RoboDK station: Rib.rdk

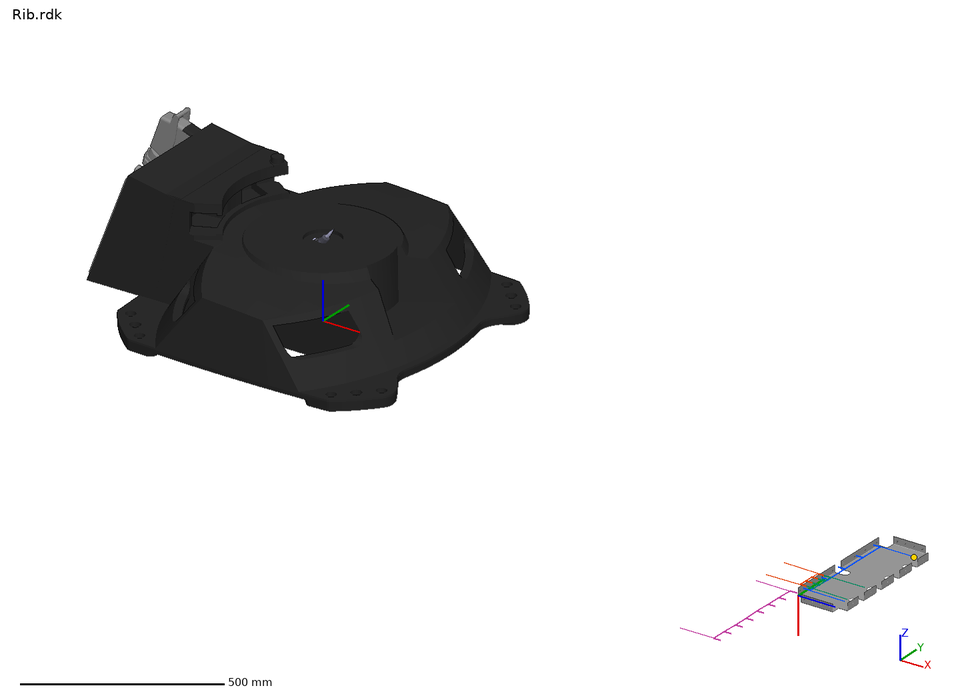
[picture v0: the station drawn from its stored meshes, robots at their saved joint values, targets as dots, program paths as lines]
Station Rib (saved by RoboDK 5.2.3). Poses are relative to the parent item; angles as X-Y-Z fixed-axis rotations.
  - frame KUKA KR 210 R2700 extra Base at (0, 0, 0) mm
    - robot KUKA KR 210 R2700 extra: 6 axes, payload 210 kg, reach 2696 mm, repeatability 0.06 mm, weight 1068 kg
        joint limits [-185, -140, -120, -350, -125, -350] to [185, -5, 155, 350, 125, 350]; home [0, -90, 90, 0, 0, 0]; saved at [-33.949, -82.089, 134.053, 57.76, 80.009, -97.195]
      - tool Spindle, TCP at (32, 0, 260) mm, rotated rx 0 ry 39 rz 0 deg, size 157.3 x 72 x 259.9 mm, geometry from Extracted Curve Point
  - frame Frame 2 at (1418.68, 0, -350) mm, rotated rx 0 ry 90 rz 0 deg
    - object rib-side at (0, 369, 0) mm, rotated rx 90 ry 0 rz 0 deg, 4 curves, geometry from Point 4
    - object rib-side at (0, -27, 0) mm, rotated rx 90 ry 0 rz 0 deg, 4 curves, geometry from Point 4
    - object rib-top at (0, 0, 146.5) mm, 5 curves, geometry from Point 5
    - object Rib at (0, 0, 0) mm, size 21.8 x 396 x 148.8 mm, geometry from Rib.stl
    - object rib-bot at (-21, 0, 0) mm, rotated rx 0 ry 0 rz 180 deg, 8 curves, geometry from Point 8
  - program target4 (36 instructions, listed below)
  - machining project Point settings: rotZ(0) | rotX(0)*rotY(0) | rotz(0) | onStart | onPathStart | onApproach | onPoint | onRetract | onFinish | SetRPM(%1) | SetTool(%1) | Extruder(%1) | default | default | OutOnMov(%1) | OutOffMov(%1) | onPathFinish | M_RunCode(%1)
  - machining project Point settings: rotZ(0) | rotX(0)*rotY(0) | rotz(0) | onStart | onPathStart | onApproach | onPoint | onRetract | onFinish | SetRPM(%1) | SetTool(%1) | Extruder(%1) | default | default | OutOnMov(%1) | OutOffMov(%1) | onPathFinish | M_RunCode(%1)
  - program target3 (31 instructions, listed below)
  - machining project Point settings: rotZ(0) | rotX(0)*rotY(0) | rotz(0) | onStart | onPathStart | onApproach | onPoint | onRetract | onFinish | SetRPM(%1) | SetTool(%1) | Extruder(%1) | default | default | OutOnMov(%1) | OutOffMov(%1) | onPathFinish | M_RunCode(%1)
  - program target1 (31 instructions, listed below)
  - machining project Point settings: rotZ(0) | rotX(0)*rotY(0) | rotz(0) | onStart | onPathStart | onApproach | onPoint | onRetract | onFinish | SetRPM(%1) | SetTool(%1) | Extruder(%1) | default | default | OutOnMov(%1) | OutOffMov(%1) | onPathFinish | M_RunCode(%1)
  - program target2 (51 instructions, listed below)
  - program MainProgram (4 instructions, listed below)
  - machining project Point settings: rotZ(0) | rotX(0)*rotY(0) | rotz(0) | onStart | onPathStart | onApproach | onPoint | onRetract | onFinish | SetRPM(%1) | SetTool(%1) | Extruder(%1) | default | default | OutOnMov(%1) | OutOffMov(%1) | onPathFinish | M_RunCode(%1)
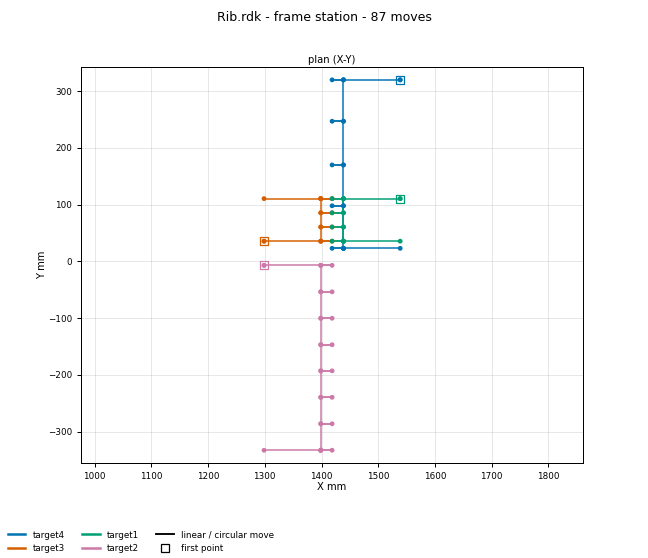
[picture p0: tool path of Rib.rdk in frame station, 87 of 87 moves have a stored position in this frame; points joined in program order, loops and branches not executed]

--- program target4 (robot KUKA KR 210 R2700 extra) ---
  Smooth(1)
  Set speed (1000.0 mm/s)
  Set Ref.: Frame 2
  Set Tool: Spindle
  Show Spindle
  MoveJ 1 to (-10, 320, 120) mm, rotated rx -180 ry 0 rz -180 deg; joints [-8.769, -14.046, 70.252, -6.836, 84.504, -4.887]
  MoveL 2 to (-10, 320, 120) mm, rotated rx -180 ry 0 rz -180 deg; joints [-8.769, -14.046, 70.252, -6.836, 84.504, -4.887]
  MoveL 3 to (-10, 320, 20) mm, rotated rx 180 ry 0 rz -180 deg; joints [-9.206, -16.545, 77.442, -7.257, 79.82, -4.534]
  MoveL 4 to (-10, 320, 20) mm, rotated rx 180 ry 0 rz -180 deg; joints [-9.206, -16.545, 77.442, -7.257, 79.82, -4.534]
  Set speed (50.0 mm/s)
  MoveL 5 to (-10, 320, 0) mm, rotated rx 180 ry 0 rz -180 deg; joints [-9.298, -16.994, 78.806, -7.352, 78.906, -4.461]
  MoveL 6 to (-10, 320, 20) mm, rotated rx 180 ry 0 rz -180 deg; joints [-9.206, -16.545, 77.442, -7.257, 79.82, -4.534]
  Set speed (1000.0 mm/s)
  MoveL 7 to (-10, 247, 20) mm, rotated rx -180 ry 0 rz -180 deg; joints [-7.13, -16.783, 78.161, -5.631, 79.454, -3.468]
  Set speed (50.0 mm/s)
  MoveL 8 to (-10, 247, 0) mm, rotated rx -180 ry 0 rz -180 deg; joints [-7.203, -17.225, 79.521, -5.706, 78.538, -3.41]
  MoveL 9 to (-10, 247, 20) mm, rotated rx -180 ry 0 rz -180 deg; joints [-7.13, -16.783, 78.161, -5.631, 79.454, -3.468]
  Set speed (1000.0 mm/s)
  MoveL 10 to (-10, 170, 20) mm, rotated rx -180 ry 0 rz -180 deg; joints [-4.921, -16.965, 78.718, -3.892, 79.168, -2.369]
  Set speed (50.0 mm/s)
  MoveL 11 to (-10, 170, 0) mm, rotated rx 180 ry 0 rz -180 deg; joints [-4.971, -17.403, 80.074, -3.944, 78.25, -2.329]
  MoveL 12 to (-10, 170, 20) mm, rotated rx -180 ry 0 rz -180 deg; joints [-4.921, -16.965, 78.718, -3.892, 79.168, -2.369]
  Set speed (1000.0 mm/s)
  MoveL 13 to (-10, 98, 20) mm, rotated rx -180 ry 0 rz -180 deg; joints [-2.841, -17.074, 79.052, -2.249, 78.996, -1.36]
  Set speed (50.0 mm/s)
  MoveL 14 to (-10, 98, 0) mm, rotated rx 180 ry 0 rz -180 deg; joints [-2.87, -17.508, 80.406, -2.28, 78.076, -1.336]
  MoveL 15 to (-10, 98, 20) mm, rotated rx -180 ry 0 rz -180 deg; joints [-2.841, -17.074, 79.052, -2.249, 78.996, -1.36]
  Set speed (1000.0 mm/s)
  MoveL 16 to (-10, 23, 20) mm, rotated rx 180 ry 0 rz -180 deg; joints [-0.667, -17.124, 79.209, -0.529, 78.915, -0.318]
  Set speed (50.0 mm/s)
  MoveL 17 to (-10, 23, 0) mm, rotated rx 180 ry 0 rz -180 deg; joints [-0.674, -17.558, 80.562, -0.536, 77.994, -0.313]
  MoveL 18 to (-10, 23, 20) mm, rotated rx 180 ry 0 rz -180 deg; joints [-0.667, -17.124, 79.209, -0.529, 78.915, -0.318]
  MoveL 19 to (-10, 23, 20) mm, rotated rx 180 ry 0 rz -180 deg; joints [-0.667, -17.124, 79.209, -0.529, 78.915, -0.318]
  Set speed (1000.0 mm/s)
  MoveL 20 to (-10, 23, 20) mm, rotated rx 180 ry 0 rz -180 deg; joints [-0.667, -17.124, 79.209, -0.529, 78.915, -0.318]
  MoveL 21 to (-10, 23, 120) mm, rotated rx -180 ry 0 rz -180 deg; joints [-0.635, -14.705, 72.09, -0.497, 83.614, -0.345]

--- program target3 (robot KUKA KR 210 R2700 extra) ---
  Smooth(1)
  Set speed (1000.0 mm/s)
  Set Ref.: Frame 2
  Set Tool: Spindle
  Show Spindle
  MoveJ 1 to (-10, 35.6, -120) mm, rotated rx 0 ry 0 rz -90 deg; joints [-36.655, -9.289, 97.989, 92.344, 89.947, -88.701]
  MoveL 2 to (-10, 35.6, -120) mm, rotated rx 0 ry 0 rz -90 deg; joints [-36.655, -9.289, 97.989, 92.344, 89.947, -88.701]
  MoveL 3 to (-10, 35.6, -20) mm, rotated rx 0 ry 0 rz -90 deg; joints [-33.402, -9.185, 100.643, 95.596, 90.142, -91.451]
  MoveL 4 to (-10, 35.6, -20) mm, rotated rx 0 ry 0 rz -90 deg; joints [-33.402, -9.185, 100.643, 95.596, 90.142, -91.451]
  Set speed (50.0 mm/s)
  MoveL 5 to (-10, 35.6, 0) mm, rotated rx 0 ry 0 rz -90 deg; joints [-32.72, -9.149, 101.134, 96.276, 90.217, -91.973]
  MoveL 6 to (-10, 35.6, -20) mm, rotated rx 0 ry 0 rz -90 deg; joints [-33.402, -9.185, 100.643, 95.596, 90.142, -91.451]
  Set speed (1000.0 mm/s)
  MoveL 7 to (-10, 60.6, -20) mm, rotated rx 0 ry 0 rz -90 deg; joints [-32.853, -9.239, 99.688, 96.147, 90.048, -90.447]
  Set speed (50.0 mm/s)
  MoveL 8 to (-10, 60.6, 0) mm, rotated rx 0 ry 0 rz -90 deg; joints [-32.177, -9.214, 100.181, 96.822, 90.115, -90.96]
  MoveL 9 to (-10, 60.6, -20) mm, rotated rx 0 ry 0 rz -90 deg; joints [-32.853, -9.239, 99.688, 96.147, 90.048, -90.447]
  Set speed (1000.0 mm/s)
  MoveL 10 to (-10, 85.6, -20) mm, rotated rx 0 ry 0 rz -90 deg; joints [-32.319, -9.275, 98.713, 96.681, 89.935, -89.442]
  Set speed (50.0 mm/s)
  MoveL 11 to (-10, 85.6, 0) mm, rotated rx 0 ry 0 rz -90 deg; joints [-31.649, -9.259, 99.205, 97.351, 89.993, -89.947]
  MoveL 12 to (-10, 85.6, -20) mm, rotated rx 0 ry 0 rz -90 deg; joints [-32.319, -9.275, 98.713, 96.681, 89.935, -89.442]
  Set speed (1000.0 mm/s)
  MoveL 13 to (-10, 110.6, -20) mm, rotated rx 0 ry 0 rz -90 deg; joints [-31.8, -9.291, 97.716, 97.197, 89.803, -88.437]
  Set speed (50.0 mm/s)
  MoveL 14 to (-10, 110.6, 0) mm, rotated rx 0 ry 0 rz -90 deg; joints [-31.136, -9.286, 98.209, 97.862, 89.853, -88.933]
  MoveL 15 to (-10, 110.6, -20) mm, rotated rx 0 ry 0 rz -90 deg; joints [-31.8, -9.291, 97.716, 97.197, 89.803, -88.437]
  MoveL 16 to (-10, 110.6, -20) mm, rotated rx 0 ry 0 rz -90 deg; joints [-31.8, -9.291, 97.716, 97.197, 89.803, -88.437]
  Set speed (1000.0 mm/s)
  MoveL 17 to (-10, 110.6, -20) mm, rotated rx 0 ry 0 rz -90 deg; joints [-31.8, -9.291, 97.716, 97.197, 89.803, -88.437]
  MoveL 18 to (-10, 110.6, -120) mm, rotated rx 0 ry 0 rz -90 deg; joints [-34.981, -9.246, 95.05, 94.009, 89.706, -85.814]

--- program target1 (robot KUKA KR 210 R2700 extra) ---
  Smooth(1)
  Set speed (1000.0 mm/s)
  Set Ref.: Frame 2
  Set Tool: Spindle
  Show Spindle
  MoveJ 1 to (-10, 110.6, 120) mm, rotated rx 180 ry 0 rz -90 deg; joints [23.134, -8.985, 102.807, -105.832, 91.044, 93.677]
  MoveL 2 to (-10, 110.6, 120) mm, rotated rx 180 ry 0 rz -90 deg; joints [23.134, -8.985, 102.807, -105.832, 91.044, 93.677]
  MoveL 3 to (-10, 110.6, 20) mm, rotated rx 180 ry 0 rz -90 deg; joints [19.166, -8.768, 104.357, -109.747, 91.894, 95.259]
  MoveL 4 to (-10, 110.6, 20) mm, rotated rx 180 ry 0 rz -90 deg; joints [19.166, -8.768, 104.357, -109.747, 91.894, 95.259]
  Set speed (50.0 mm/s)
  MoveL 5 to (-10, 110.6, 0) mm, rotated rx 180 ry 0 rz -90 deg; joints [18.348, -8.723, 104.629, -110.552, 92.08, 95.528]
  MoveL 6 to (-10, 110.6, 20) mm, rotated rx 180 ry 0 rz -90 deg; joints [19.166, -8.768, 104.357, -109.747, 91.894, 95.259]
  Set speed (1000.0 mm/s)
  MoveL 7 to (-10, 85.6, 20) mm, rotated rx -180 ry 0 rz -90 deg; joints [19.526, -8.595, 105.346, -109.349, 92.246, 96.369]
  Set speed (50.0 mm/s)
  MoveL 8 to (-10, 85.6, 0) mm, rotated rx 180 ry 0 rz -90 deg; joints [18.695, -8.542, 105.617, -110.163, 92.45, 96.64]
  MoveL 9 to (-10, 85.6, 20) mm, rotated rx -180 ry 0 rz -90 deg; joints [19.526, -8.595, 105.346, -109.349, 92.246, 96.369]
  Set speed (1000.0 mm/s)
  MoveL 10 to (-10, 60.6, 20) mm, rotated rx 180 ry 0 rz -90 deg; joints [19.9, -8.396, 106.314, -108.931, 92.584, 97.487]
  Set speed (50.0 mm/s)
  MoveL 11 to (-10, 60.6, 0) mm, rotated rx -180 ry 0 rz -90 deg; joints [19.055, -8.335, 106.585, -109.755, 92.806, 97.761]
  MoveL 12 to (-10, 60.6, 20) mm, rotated rx 180 ry 0 rz -90 deg; joints [19.9, -8.396, 106.314, -108.931, 92.584, 97.487]
  Set speed (1000.0 mm/s)
  MoveL 13 to (-10, 35.6, 20) mm, rotated rx 180 ry 0 rz -90 deg; joints [20.287, -8.172, 107.26, -108.494, 92.905, 98.616]
  Set speed (50.0 mm/s)
  MoveL 14 to (-10, 35.6, 0) mm, rotated rx 180 ry 0 rz -90 deg; joints [19.429, -8.102, 107.531, -109.327, 93.146, 98.893]
  MoveL 15 to (-10, 35.6, 20) mm, rotated rx 180 ry 0 rz -90 deg; joints [20.287, -8.172, 107.26, -108.494, 92.905, 98.616]
  MoveL 16 to (-10, 35.6, 20) mm, rotated rx 180 ry 0 rz -90 deg; joints [20.287, -8.172, 107.26, -108.494, 92.905, 98.616]
  Set speed (1000.0 mm/s)
  MoveL 17 to (-10, 35.6, 20) mm, rotated rx 180 ry 0 rz -90 deg; joints [20.287, -8.172, 107.26, -108.494, 92.905, 98.616]
  MoveL 18 to (-10, 35.6, 120) mm, rotated rx 180 ry 0 rz -90 deg; joints [24.437, -8.522, 105.716, -104.454, 91.804, 96.965]

--- program target2 (robot KUKA KR 210 R2700 extra) ---
  Smooth(1)
  Set speed (1000.0 mm/s)
  Set Ref.: Frame 2
  Set Tool: Spindle
  Show Spindle
  MoveJ 1 to (-10, -7, -120) mm; joints [-0.441, -16.759, 131.622, 179.647, 75.862, -0.191]
  MoveL 2 to (-10, -7, -120) mm; joints [-0.441, -16.759, 131.622, 179.647, 75.862, -0.191]
  MoveL 3 to (-10, -7, -20) mm; joints [-0.397, -19.457, 128.225, 179.671, 69.767, -0.136]
  MoveL 4 to (-10, -7, -20) mm; joints [-0.397, -19.457, 128.225, 179.671, 69.767, -0.136]
  Set speed (50.0 mm/s)
  MoveL 5 to (-10, -7, 0) mm; joints [-0.39, -19.904, 127.502, 179.675, 68.598, -0.127]
  MoveL 6 to (-10, -7, -20) mm; joints [-0.397, -19.457, 128.225, 179.671, 69.767, -0.136]
  Set speed (1000.0 mm/s)
  MoveL 7 to (-10, -53.67, -20) mm; joints [-3.044, -19.489, 128.175, 177.478, 69.664, -1.039]
  Set speed (50.0 mm/s)
  MoveL 8 to (-10, -53.67, 0) mm; joints [-2.985, -19.933, 127.451, 177.507, 68.499, -0.965]
  MoveL 9 to (-10, -53.67, -20) mm; joints [-3.044, -19.489, 128.175, 177.478, 69.664, -1.039]
  Set speed (1000.0 mm/s)
  MoveL 10 to (-10, -100.33, -20) mm; joints [-5.676, -19.57, 128.047, 175.29, 69.403, -1.919]
  Set speed (50.0 mm/s)
  MoveL 11 to (-10, -100.33, 0) mm; joints [-5.567, -20.008, 127.324, 175.344, 68.249, -1.781]
  MoveL 12 to (-10, -100.33, -20) mm; joints [-5.676, -19.57, 128.047, 175.29, 69.403, -1.919]
  Set speed (1000.0 mm/s)
  MoveL 13 to (-10, -147, -20) mm; joints [-8.286, -19.698, 127.842, 173.11, 68.989, -2.756]
  Set speed (50.0 mm/s)
  MoveL 14 to (-10, -147, 0) mm; joints [-8.127, -20.125, 127.119, 173.188, 67.853, -2.557]
  MoveL 15 to (-10, -147, -20) mm; joints [-8.286, -19.698, 127.842, 173.11, 68.989, -2.756]
  Set speed (1000.0 mm/s)
  MoveL 16 to (-10, -193, -20) mm; joints [-10.824, -19.866, 127.565, 170.971, 68.44, -3.52]
  Set speed (50.0 mm/s)
  MoveL 17 to (-10, -193, 0) mm; joints [-10.619, -20.279, 126.842, 171.071, 67.328, -3.264]
  MoveL 18 to (-10, -193, -20) mm; joints [-10.824, -19.866, 127.565, 170.971, 68.44, -3.52]
  Set speed (1000.0 mm/s)
  MoveL 19 to (-10, -239.67, -20) mm; joints [-13.357, -20.075, 127.207, 168.815, 67.749, -4.217]
  Set speed (50.0 mm/s)
  MoveL 20 to (-10, -239.67, 0) mm; joints [-13.106, -20.47, 126.484, 168.935, 66.666, -3.906]
  MoveL 21 to (-10, -239.67, -20) mm; joints [-13.357, -20.075, 127.207, 168.815, 67.749, -4.217]
  Set speed (1000.0 mm/s)
  MoveL 22 to (-10, -286.33, -20) mm; joints [-15.837, -20.317, 126.772, 166.673, 66.935, -4.819]
  Set speed (50.0 mm/s)
  MoveL 23 to (-10, -286.33, 0) mm; joints [-15.544, -20.692, 126.049, 166.811, 65.885, -4.46]
  MoveL 24 to (-10, -286.33, -20) mm; joints [-15.837, -20.317, 126.772, 166.673, 66.935, -4.819]
  Set speed (1000.0 mm/s)
  MoveL 25 to (-10, -333, -20) mm; joints [-18.258, -20.587, 126.26, 164.545, 66.012, -5.315]
  Set speed (50.0 mm/s)
  MoveL 26 to (-10, -333, 0) mm; joints [-17.926, -20.939, 125.538, 164.697, 64.999, -4.91]
  MoveL 27 to (-10, -333, -20) mm; joints [-18.258, -20.587, 126.26, 164.545, 66.012, -5.315]
  MoveL 28 to (-10, -333, -20) mm; joints [-18.258, -20.587, 126.26, 164.545, 66.012, -5.315]
  Set speed (1000.0 mm/s)
  MoveL 29 to (-10, -333, -20) mm; joints [-18.258, -20.587, 126.26, 164.545, 66.012, -5.315]
  MoveL 30 to (-10, -333, -120) mm; joints [-20.111, -18.447, 129.662, 163.602, 71.18, -7.554]

--- program MainProgram (robot KUKA KR 210 R2700 extra) ---
  Call target1
  Call target2
  Call target3
  Call target4
